// TwinCAT 3 PLC project FourceAutomotivePLC
// ProgramVersion: 3.1.4024.0
// libraries:
//   Tc2_Standard, * (Beckhoff Automation GmbH)
//   Tc2_System, * (Beckhoff Automation GmbH)
//   Tc3_Module, * (Beckhoff Automation GmbH)
//   VisuSymbols,3.5.10.0,System
// project tree:
//   DUTs/ Task_1.TcDUT, Task_2.TcDUT
//   / GlobalTextList.TcGTLO, PlcTask.TcTTO, TASK_1_1.TcTTO, Visualization Manager.TcVMO (not stored)
//   GVLs/ GVL_FourceAutomotive.TcGVL
//   POUs/ Controleren_tijd.TcPOU, MAIN.TcPOU, Orderverwerking_magazijn.TcPOU, POU.TcPOU (not stored), Transporteren_order.TcPOU
//   VISUs/ FouceAutomotiveVisualisation.TcVIS, Visualization.TcVIS
// real-time tasks:
//   TASK PlcTask: cycle T#10ms, priority 20, ADS port 350
//   TASK TASK_1: cycle T#10ms, priority 1, ADS port 351

CONFIGURATION FourceAutomotivePLC
    RESOURCE PLC ON TwinCAT3
        TASK PlcTask(INTERVAL := T#10ms, PRIORITY := 20);
        TASK TASK_1_1(INTERVAL := T#10ms, PRIORITY := 1);
        PROGRAM MAIN WITH PlcTask : MAIN;
    END_RESOURCE
END_CONFIGURATION

// ---- DUTs/Task_1.TcDUT
TYPE Task_1 :
	(
		NieuweOrderGaragist,
		VoorraadAdministratief,
		VerzamelingArtikelen,
		OrderGeanuleerd
	) := NieuweOrderGaragist;
END_TYPE

// ---- DUTs/Task_2.TcDUT
TYPE Task_2 :
(
		Inladen,
		Transport,
		Afleveren
	) := Inladen;
END_TYPE

// ---- GVLs/GVL_FourceAutomotive.TcGVL
{attribute 'qualified_only'}
VAR_GLOBAL
	currentState : Task_1 := Task_1.NieuweOrderGaragist;   
	Nieuwe_order: BOOL := TRUE;
	Controleren_voorraad: INT := 0;
	Order_magazijn: BOOL;
	Order_uitgeprint: BOOL;
	Order_verzameld: BOOL; 
	Geannuleerd: BOOL;
	Order_controle: INT :=0;
	Order_voltooid: BOOL;
END_VAR

// ---- POUs/MAIN.TcPOU
PROGRAM MAIN
VAR
	currentState : Task_1 := Task_1.NieuweOrderGaragist;   
	Nieuwe_order: BOOL := TRUE;
	Controleren_voorraad: INT := 0;
	Order_magazijn: BOOL;
	Order_uitgeprint: BOOL;
	Order_verzameld: BOOL; 
	Geannuleerd: BOOL;
	Order_controle: INT :=0;
	Order_voltooid: BOOL;
END_VAR

END_PROGRAM

// ---- POUs/Controleren_tijd.TcPOU
FUNCTION Controleren_tijd : BOOL
VAR
  Huidige_tijd : INT; //Invoer van de tijd
END_VAR

IF (Huidige_tijd >= 0) AND (Huidige_tijd <= 2400) THEN
	IF Huidige_tijd >= 1000 THEN
		Controleren_tijd := TRUE
	ELSIF
		Controleren_tijd := FALSE
	END_IF
ELSE
	Controleren_tijd := FALSE //Geeft aan dat de ingevoerde tijd ongeldig is
END_IF;

END_FUNCTION

// ---- POUs/Orderverwerking_magazijn.TcPOU
PROGRAM Orderverwerking_magazijn
VAR
	currentState : Task_1 := Task_1.NieuweOrderGaragist;   
	Nieuwe_order: BOOL := TRUE;
	Controleren_voorraad: INT := 0;
	Order_magazijn: BOOL;
	Order_uitgeprint: BOOL;
	Order_verzameld: BOOL; 
	Geannuleerd: BOOL;
	Order_controle: INT :=0;
	Order_voltooid: BOOL;
END_VAR

CASE currentState OF
    Task_1.NieuweOrderGaragist:
        // Nieuwe bestelling van een garagist
        IF Nieuwe_order = TRUE THEN
            currentState := VoorraadAdministratief;
        END_IF;
		
	Task_1.VoorraadAdministratief:
		// Controleren of de voorraad klopt (Adminastratief)
		IF Controleren_voorraad = 1 THEN
			Order_magazijn := TRUE;
			Order_uitgeprint := TRUE;
			Order_verzameld := TRUE;
			Geannuleerd := FALSE;
			currentState := VerzamelingArtikelen;
		ELSIF Controleren_voorraad = 2 THEN
			Order_magazijn := FALSE;
			Order_uitgeprint := FALSE;
			Order_verzameld := FALSE;
			Geannuleerd := TRUE;
		END_IF
	
		
	Task_1.VerzamelingArtikelen:
	// Controleren of de verzamelde artikelen overeenkomen met de Orderverzamellijst
		IF Order_controle = 1 THEN
			Order_voltooid := TRUE;
			Geannuleerd := FALSE;
		ELSIF Order_controle = 2 THEN
			Order_controle := 0;
			Order_voltooid := FALSE;
			Geannuleerd := FALSE;
		ELSIF Order_controle = 3 THEN
			Order_voltooid := FALSE;
			Geannuleerd := TRUE;			
		END_IF
		
END_CASE;

END_PROGRAM

// ---- POUs/Transporteren_order.TcPOU
PROGRAM Transporteren_order
VAR
	currentState : Taks_2 : Task_2.Inladen;
	
	Result: INT;
	IsTimeGreaterThan10: INT;
	UserInputTime: INT;
END_VAR

END_PROGRAM

// ---- GlobalTextList.TcGTLO
TEXTLIST GlobalTextList
  768 = 'Nieuwe_order'
END_TEXTLIST

// ---- VISUs/FouceAutomotiveVisualisation.TcVIS
VISUALIZATION FouceAutomotiveVisualisation  // 2x2
END_VISUALIZATION

// ---- VISUs/Visualization.TcVIS
VISUALIZATION Visualization  // 2x2
END_VISUALIZATION
